# EPICS substitutions: src/main/epics/hnossApp/Db/hnoss.substitutions
#HNOSS

file "DI.template" { pattern

#PSL SUBS?
{SUBS,	DEV,       OFFS,   OFFS2}
{Rhtr,	LS550,      84,	    84}
{PSL,	PSL,        86,     86}
}

file "AI.template" { pattern

#unsure about units..
{SUBS,	DEV,       OFFS,   OFFS2, LOPR, HOPR, EGU}
{LHe,	TT140A,   130,	   130,	  0,	500,   K}
{LHe,	TT140B,   136,	   136,	  0,	500,   K}
{LHe,   TT140C,   142,     142,   0,    500,   K}
{LHe,   TT140D,   148,     148,   0,    500,   K}
{LHe,   TT141,    154,     154,   0,    500,   K}
{LHe,   TT142A,   160,     160,   0,    500,   K}
{LHe,   TT142B,   166,     166,   0,    500,   K}
{LHe,   TT143A,   172,     172,   0,    500,   K}
{LHe,   TT143B,   178,     178,   0,    500,   K}
{LHe,   TT143C,   184,     184,   0,    500,   K}
{LHe,   TT144A,   190,     190,   0,    500,   K}
{LHe,   TT144B,   196,     196,   0,    500,   K}
{LHe,   TT144C,   202,     202,   0,    500,   K}
{LHe,   TT145A,   208,     208,   0,    500,   K}
{LHe,   TT145B,   214,     214,   0,    500,   K}
{LHe,   TT146A,   220,     220,   0,    500,   K}
{LHe,   TT146B,   226,     226,   0,    500,   K}
{LHe,   TT147,    232,     232,   0,    500,   K}
{LHe,   TT148,    238,     238,   0,    500,   K}
{LN2,   TT200,    244,     244,   0,    500,   K}
{LN2,   TT201,    250,     250,   0,    500,   K}
{LN2,   TT202,    256,     256,   0,    500,   K}
{LN2,   TT203,    262,     262,   0,    500,   K}
{LN2,   TT204,    268,     268,   0,    500,   K}
{LN2,   TT205,    274,     274,   0,    500,   K}
{LN2,   TT206,    280,     280,   0,    500,   K}
{LN2,   TT207,    286,     286,   0,    500,   K}
{LN2,   TT208,    292,     292,   0,    500,   K}
{LN2,   TT209,    298,     298,   0,    500,   K}
{LN2,   TT210,    304,     304,   0,    500,   K}
{LN2,   TT211,    310,     310,   0,    500,   K}
{LN2,   TT212,    316,     316,   0,    500,   K}
{LN2,   TT213,    322,     322,   0,    500,   K}
{LN2,   TT214A,   328,     328,   0,    500,   K}
{LN2,   TT214B,   334,     334,   0,    500,   K}
{LN2,   TT214C,   340,     340,   0,    500,   K}
{LN2,   TT215,    346,     346,   0,    500,   K}
{LN2,   TT216A,   352,     352,   0,    500,   K}
{LN2,   TT216B,   358,     358,   0,    500,   K}
{LN2,   TT216C,   364,     364,   0,    500,   K}
{LN2,   TT216D,   370,     370,   0,    500,   K}
{LN2,   TT216E,   376,     376,   0,    500,   K}
{LN2,   TT216F,   382,     382,   0,    500,   K}
{LN2,   TT217,    388,     388,   0,    500,   K}
{SHe,   TT300,    394,     394,   0,    500,   K}
{SHe,   TT307,    400,     400,   0,    500,   K}
{SHe,   TT308,    406,     406,   0,    500,   K}
{SHe,   TT309,    412,     412,   0,    500,   K}
{SHe,   TT310,    418,     418,   0,    500,   K}
{SHe,   TT311,    424,     424,   0,    500,   K}
{SHe,   TT312,    430,     430,   0,    500,   K}
{IBoxN2,TT400,    436,     436,   0,    500,   K}
{IBoxN2,TT401A,   442,     442,   0,    500,   K}
{IBoxN2,TT401B,   448,     448,   0,    500,   K}
{IBoxN2,TT401C,   454,     454,   0,    500,   K}
{IBoxN2,TT402,    460,     460,   0,    500,   K}
{IBoxN2,TT403,    466,     466,   0,    500,   K}
{IBoxN2,TT404,    472,     472,   0,    500,   K}
{IBoxN2,TT405,    478,     478,   0,    500,   K}
{RHtr,  TT550,    484,     484,   0,    500,   K}
{SHe,   PT300,    490,     490,   0,    500,   Pa}
{SHe,   PT301,    496,     496,   0,    500,   Pa}
{SHe,   PT302,    502,     502,   0,    500,   Pa}
{IBoxHe,PT500,    508,     508,   0,    500,   Pa}
{LN2,   PT200,    514,     514,   0,    500,   Pa}
{LHe,   LT100,    520,     520,   0,    500,   m}
{LHe,   LT101,    526,     526,   0,    500,   m}
{LN2,   FT200,    532,     532,   0,    500,   m3/s}
{LN2,   FT201,    538,     538,   0,    500,   m3/s}
{LN2,   FT202,    544,     544,   0,    500,   m3/s}
{SHe,   FT301,    550,     550,   0,    500,   m3/s}
{SHe,   FT302,    556,     556,   0,    500,   m3/s}
{RHtr,  FT550,    562,     562,   0,    500,   m3/s}
{RHtr,  FT551,    568,     568,   0,    500,   m3/s}
{RHtr,  FT552,    574,     574,   0,    500,   m3/s}
{LHe,   TT100,    706,     706,   0,    500,   K}
{LHe,   TT101,    712,     712,   0,    500,   K}
{LHe,   TT102,    718,     718,   0,    500,   K}
{LHe,   TT103,    724,     724,   0,    500,   K}
{LHe,   TT104,    730,     730,   0,    500,   K}
{LHe,   TT105,    736,     736,   0,    500,   K}
{LHe,   TT106,    742,     742,   0,    500,   K}
{LHe,   TT107,    748,     748,   0,    500,   K}
{LHe,   TT108,    754,     754,   0,    500,   K}
{LHe,   TT109,    760,     760,   0,    500,   K}
{LHe,   TT110,    766,     766,   0,    500,   K}
{LHe,   TT111,    772,     772,   0,    500,   K}
{LHe,   TT112,    778,     778,   0,    500,   K}
{LHe,   TT113,    784,     784,   0,    500,   K}
{LHe,   TT114,    790,     790,   0,    500,   K}
{LHe,   TT115,    796,     796,   0,    500,   K}
{LHe,   TT116,    802,     802,   0,    500,   K}
{LHe,   TT117,    808,     808,   0,    500,   K}
{LHe,   TT118,    814,     814,   0,    500,   K}
{LHe,   TT119,    820,     820,   0,    500,   K}
{LHe,   TT120,    826,     826,   0,    500,   K}
{LHe,   TT121,    832,     832,   0,    500,   K}
{LHe,   TT122,    838,     838,   0,    500,   K}
{LHe,   TT123,    844,     844,   0,    500,   K}
{LHe,   TT124,    850,     850,   0,    500,   K}
{LHe,   TT125,    856,     856,   0,    500,   K}
{LHe,   TT126,    862,     862,   0,    500,   K}
{LHe,   TT127,    868,     868,   0,    500,   K}
{LHe,   TT128,    874,     874,   0,    500,   K}
{LHe,   TT129,    880,     880,   0,    500,   K}
{LHe,   TT130,    886,     886,   0,    500,   K}
{SHe,   TT301,    892,     892,   0,    500,   K}
{SHe,   TT302,    898,     898,   0,    500,   K}
{SHe,   TT303,    904,     904,   0,    500,   K}
{SHe,   TT304,    910,     910,   0,    500,   K}
{SHe,   TT305,    916,     916,   0,    500,   K}
{SHe,   TT306,    922,     922,   0,    500,   K}
{IBoxHe,TT500,    928,     928,   0,    500,   K}
{IBoxHe,TT501,    934,     934,   0,    500,   K}
{IBoxHe,TT502,    940,     940,   0,    500,   K}
{RHtr,  PT551,   1072,    1072,   0,    500,   Pa}
{RHtr,  PT552,   1078,    1078,   0,    500,   Pa}
{LHe,   PT100,   1084,    1084,   0,    500,   Pa}
{RHtr,  PT550,   1090,    1090,   0,    500,   Pa}
{LHe,   PT101,   1096,    1096,   0,    500,   Pa}
{LHe,   PT102,   1102,    1102,   0,    500,   Pa}
{Vac,   PT000,   1234,    1234,   0,    500,   Pa}
{Vac,   PT001,   1240,    1240,   0,    500,   Pa}
{Vac,   PT002,   1246,    1246,   0,    500,   Pa}
{Vac,   PT003,   1252,    1252,   0,    500,   Pa}
{Vac,   PT004,   1258,    1258,   0,    500,   Pa}
}

file "Valves.template" { pattern
{SUBS,	DEV,       OFFS,   OFFS2}
{Vac,	FV000,     1438,    1438}
{Vac,	FV001,     1440,    1440}
{Vac,	FV010,     1442,    1442}
{Vac,	FV011,     1444,    1444}
{Vac,	FV012,     1446,    1446}
{LHe,	FV100,     1448,    1448}
{LHe,	FV101,     1450,    1450}
{LN2,	FV200,     1452,    1452}
{SHe,	FV300,     1454,    1454}
{SHe,	FV301,     1456,    1456}
{SHe,	FV302,     1458,    1458}
{IBoxN2,FV400,     1460,    1460}
{IBoxN2,FV401,     1462,    1462}
{IBoxHe,FV500,     1464,    1464}
{IBoxHe,FV501,     1466,    1466}
{IBoxHe,FV502,     1468,    1468}
{RHtr,  FV550,     1470,    1470}
{RHtr,  FV551,     1472,    1472}
}

file "Evalves.template" { pattern
{SUBS,	DEV,       OFFS,   OFFS2}
{LN2,	EV200,     1390,    1390}
{LN2,	EV201,     1392,    1392}
{IBoxN2,EV400,     1394,    1394}
}

file "AValves.template" { pattern
{SUBS,	DEV,       OFFS,   OFFS2, LOPR, HOPR, EGU}
{LHe,	CV100,   1516,	   1516,   0,	100,  percent}
{LHe,	CV101,   1522,	   1522,   0,	100,  percent}
{LHe,	CV102,   1528,	   1528,   0,	100,  percent}
{LHe,	CV103,   1534,	   1534,   0,	100,  percent}
{LHe,	CV104,   1540,	   1540,   0,	100,  percent}
{LHe,	CV105,   1546,	   1546,   0,	100,  percent}
{LN2,	CV200,   1552,	   1552,   0,	100,  percent}
{LN2,	CV201,   1558,	   1558,   0,	100,  percent}
{SHe,	CV301,   1564,	   1564,   0,	100,  percent}
{SHe,	CV302,   1570,	   1570,   0,	100,  percent}
{RHtr,	CV550,   1576,	   1576,   0,	100,  percent}
{RHtr,	CV551,   1582,	   1582,   0,	100,  percent}
{RHtr,	CV552,   1588,	   1588,   0,	100,  percent}
}

file "PID.template" { pattern
{SUBS,   DEV,     OFFS,   OFFS2,    EGU}
{LN2,    TIC200,  1720,   1720,    unknown}
{LN2,    FIC200,  1742,   1730,    unknown}
{LN2,    TIC201,  1764,   1740,    unknown}
{LN2,    FIC201,  1786,   1750,    unknown}
{SHe,    TIC301,  1808,   1760,    unknown}
{SHe,    FIC301,  1830,   1770,    unknown}
{SHe,    TIC302,  1852,   1780,    unknown}
{SHe,    FIC302,  1874,   1790,    unknown}
{LHe,    TIC101,  1896,   1800,    unknown}
{MKS,    MKS1,    1918,   1810,    unknown}
{MKS,    MKS2,    1940,   1820,    unknown}
{MKS,    MKS3,    1962,   1830,    unknown}
}

file "Heater1.template" { pattern
{SUBS,	DEV,       OFFS,   OFFS2}
{LHe,	EH100,     2446,    2050}
{LHe,	EH101,     2456,    2060}
{LHe,	EH102,     2466,    2070}
{LHe,	EH103,     2476,    2080}
{LHe,	EH104,     2486,    2090}
{LHe,	EH105,     2496,    2100}
{LHe,	EH106,     2506,    2110}
{LHe,	EH107,     2516,    2120}
{LHe,	EH108,     2526,    2130}
{LN2,	EH200,     2536,    2140}
{LN2,	EH201,     2546,    2150}
{LN2,	EH202,     2556,    2160}
{LN2,	EH203,     2566,    2170}
{LN2,	EH204,     2576,    2180}
{LN2,	EH205,     2586,    2190}
{LN2,	EH206,     2596,    2200}
{LN2,	EH207,     2606,    2210}
{LN2,	EH208,     2616,    2220}
{SHe,	EH300,     2626,    2230}
{SHe,	EH301,     2636,    2240}
{SHe,	EH302,     2646,    2250}
{SHe,	EH303,     2656,    2260}
{IBoxN2,EH400,     2666,    2270}
{IBoxN2,EH401,     2676,    2280}
}

file "Heater2.template" { pattern
{SUBS,	DEV,       OFFS,   OFFS2}
{Rhtr,	EH550,     2896,    2500}
}

file "SQbinary.template" { pattern
{SUBS, OFFS2, OFFS}
{SQ0,   2808, 3204}
{SQ1,   2892, 3306}
{SQ2,   2976, 3408}
{SQ3A,  3060, 3510}
{SQ3B,  3144, 3612}
{SQ4,   3228, 3714}
{SQ5,   3312, 3816}
{SQ6,   3396, 3918}
{SQ7,   3480, 4020}
{SQ8,   3564, 4122}
{SQ9,   3648, 4224}
{SQ10,  3732, 4326}
{SQ11,  3816, 4428}
{SQ12A, 3900, 4530}
{SQ12B, 3984, 4632}
{SQ13,  4068, 4734}
{SQ20,  4152, 4836}
}

file "SQanalog.template" { pattern
{SUBS,	 SIG,          OFFS2, TYPE, SIG2,	OFFS, EGU}
{SQ0,	cNcycle,       2810, INT16, sNcycle, 3224, ""}
{SQ0,	cVacRate,      2812, INT16, sVacRate, 3226,	"s"}
{SQ0,	cPressRate,    2814, INT16, sPressRate, 3228,	"s"}
{SQ0,	cVacRateAlrm,  2816, INT16, sVacRateAlrm, 3230,	"s"}
{SQ0,	cPresRateAlrm, 2818, INT16, sPresRateAlrm, 3232,"s"}
{SQ0,	cVac,          2828, FLOAT, sVac, 3242,	   "mbar"}
{SQ0,	cVacFlt,       2832, FLOAT, sVacFlt, 3246, "mbar"}
{SQ0,	cPressEOF,     2836, FLOAT, sPressEOF, 3250, "mbar"}
{SQ0,	cPressFlt,     2840, FLOAT, sPressFlt, 3254, "mbar"}
{SQ1,	cNcycle,       2894, INT16, sNcycle, 3326,   ""}
{SQ1,	cVacRate,      2896, INT16, sVacRate, 3328,  "s"}
{SQ1,	cPressRate,    2898, INT16, sPressRate, 3330,	"s"}
{SQ1,	cVacRateAlrm,  2900, INT16, sVacRateAlrm, 3332,	"s"}
{SQ1,	cPresRateAlrm, 2902, INT16, sPresRateAlrm, 3334,	"s"}
{SQ1,	cVac,          2912, FLOAT, sVac, 3344,	   "mbar"}
{SQ1,	cVacFlt,       2916, FLOAT, sVacFlt, 3348,	   "mbar"}
{SQ1,	cPressEOF,     2920, FLOAT, sPressEOF, 3352,	   "mbar"}
{SQ1,	cPressFlt,     2924, FLOAT, sPressFlt, 3356,	   "mbar"}
{SQ1,	cP_CV100,      2928, FLOAT, sP_CV100, 3360,   ""}
{SQ1,	cP_CV101,      2932, FLOAT, sP_CV101, 3364,   ""}
{SQ1,	cP_CV102,      2936, FLOAT, sP_CV102, 3368,   ""}
{SQ1,	cP_CV103,      2940, FLOAT, sP_CV103, 3372,   ""}
{SQ1,	cP_CV104,      2944, FLOAT, sP_CV104, 3376,   ""}
{SQ1,	cP_CV105,      2948, FLOAT, sP_CV105, 3380,   ""}
{SQ1,	cP_CV550,      2952, FLOAT, sP_CV550, 3384,   ""}
{SQ1,	cP_CV551,      2956, FLOAT, sP_CV551, 3388,   ""}
{SQ2,	cNcycle,       2978, INT16, sNcycle, 3428,   ""}
{SQ2,	cVacRate,      2980, INT16, sVacRate, 3430	"s"}
{SQ2,	cPressRate,    2982, INT16, sPressRate, 3432	"s"}
{SQ2,	cVacRateAlrm,  2984, INT16, sVacRateAlrm, 3434	"s"}
{SQ2,	cPresRateAlrm, 2986, INT16, sPresRateAlrm, 3436	"s"}
{SQ2,	cVac,          2996, FLOAT, sVac, 3446	"mbar"}
{SQ2,	cVacFlt,       3000, FLOAT, sVacFlt, 3450	"mbar"}
{SQ2,	cPressEOF,     3004, FLOAT, sPressEOF, 3454	"mbar"}
{SQ2,	cPressFlt,     3008, FLOAT, sPressFlt, 3458	"mbar"}
{SQ2,	cP_CV301,      3012, FLOAT, sP_CV301, 3462	""}
{SQ2,	cP_CV302,      3016, FLOAT, sP_CV302, 3466	""}
{SQ3A,	cP_Tt,         3080, FLOAT, sP_Tt, 3548	""}
{SQ3A,	cP_Low_Tt,     3084, FLOAT, sP_Low_Tt, 3552	""}
{SQ3A,	cP_High_Tt,    3088, FLOAT, sP_High_Tt, 3556	""}
{SQ3B,	cP_Tt,         3164, FLOAT, sP_Tt, 3650	""}
{SQ3B,	cP_Low_Tt,     3168, FLOAT, sP_Low_Tt, 3654	""}
{SQ3B,	cP_High_Tt,    3172, FLOAT, sP_High_Tt, 3658	""}
{SQ4,	cP_CV200_Tt,   3248, FLOAT, sP_CV200_Tt, 3752	""}
{SQ4,	cP_CV200_Ft,   3252, FLOAT, sP_CV200_Ft, 3756	""}
{SQ4,	cP_CV201_Tt,   3256, FLOAT, sP_CV201_Tt, 3760	""}
{SQ4,	cP_CV201_Ft,   3260, FLOAT, sP_CV201_Ft, 3764	""}
{SQ5,	cP_PT,         3332,  FLOAT, sP_PT,      3854	""}
{SQ5,	cP_FT,         3336,  FLOAT, sP_FT,      3858	""}
{SQ5,	cP_CV550,      3340,  FLOAT, sP_CV550,   3862	""}
{SQ5,	cP_LowLt,      3344,  FLOAT, sP_LowLt,   3866	""}
{SQ5,	cP_CoolD_Tt,   3348,  FLOAT, sP_CoolD_Tt,3870	""}
{SQ5,	cP_HighLt,     3352,  FLOAT, sP_HighLt,  3874	""}
{SQ5,	cP_CV100,      3356,  FLOAT, sP_CV100,   3878	""}
{SQ6,	cP_Tt,         3416,  FLOAT, sP_Tt,      3956	""}
{SQ6,	cP_Lt,         3420,  FLOAT, sP_Lt,      3960	""}
{SQ7,	cP_PT,         3500,  FLOAT, sP_PT,      4058	""}
{SQ7,	cP_FT550,      3504,  FLOAT, sP_FT550,   4062	""}
{SQ7,	cP_Tt_Cold,    3508,  FLOAT, sP_Tt_Cold, 4066	""}
{SQ7,	cP_SP_Tt,      3512,  FLOAT, sP_SP_Tt,   4070	""}
{SQ7,	cP_CV550,      3516,  FLOAT, sP_CV550,   4074	""}
{SQ7,	cP_CV551,      3520,  FLOAT, sP_CV551,   4078	""}
{SQ7,	cP_FT552,      3524,  FLOAT, sP_FT552,   4082	""}
{SQ7,	cP_HighLt,     3528,  FLOAT, sP_HighLt,  4086	""}
{SQ7,	cP_LowLt,      3532,  FLOAT, sP_LowLt,   4090	""}
{SQ7,	cP_CV552,      3536,  FLOAT, sP_CV552,   4094	""}
{SQ7,	cP_CV101,      3540,  FLOAT, sP_CV101,   4098	""}
{SQ7,	cP_CV102,      3544,  FLOAT, sP_CV102,   4102	""}
{SQ7,	cP_CV103,      3548,  FLOAT, sP_CV103,   4106	""}
{SQ7,	cP_CV104,      3552,  FLOAT, sP_CV104,   4110	""}
{SQ8,	cP_CV550,      3584,  FLOAT, sP_CV550,   4160	""}
{SQ8,	cP_LowLt,      3588,  FLOAT, sP_LowLt,   4164	""}
{SQ8,	cP_HighLt,     3592,  FLOAT, sP_HighLt,  4168	""}
{SQ8,	cP_Pt,         3596,  FLOAT, sP_Pt,      4172	""}
{SQ8,	cP_SP_Tt,      3600,  FLOAT, sP_SP_Tt,   4176	""}
{SQ8,	cP_CV551,      3604,  FLOAT, sP_CV551,   4180	""}
{SQ8,	cP_CV552,      3608,  FLOAT, sP_CV552,   4184	""}
{SQ8,	cP_CV104,      3612,  FLOAT, sP_CV104,   4188	""}
{SQ9,	cP_CV550,      3668,  FLOAT, sP_CV550,   4262	""}
{SQ9,	cP_LowLt,      3672,  FLOAT, sP_LowLt,   4266	""}
{SQ9,	cP_HighLt,     3676,  FLOAT, sP_HighLt,  4270	""}
{SQ9,	cP_Pt,         3680,  FLOAT, sP_Pt,      4274	""}
{SQ9,	cP_SP_Tt,      3684,  FLOAT, sP_SP_Tt,   4278	""}
{SQ9,	cP_CV105,      3688,  FLOAT, sP_CV105,   4282	""}
{SQ9,	cP_CV551_Reg,  3692,  FLOAT, sP_CV551_Reg,4286	""}
{SQ9,	cP_Final_Pt,   3696,  FLOAT, sP_Final_Pt,4290	""}
{SQ9,	cP_CV551_Pt00, 4740,  FLOAT, sP_CV551_Pt00,5550	""}
{SQ9,	cP_CV551_Pt01, 4744,  FLOAT, sP_CV551_Pt01,5554	""}
{SQ9,	cP_CV551_Pt02, 4748,  FLOAT, sP_CV551_Pt02,5558	""}
{SQ9,	cP_CV551_Pt03, 4752,  FLOAT, sP_CV551_Pt03,5562	""}
{SQ9,	cP_CV551_Pt04, 4756,  FLOAT, sP_CV551_Pt04,5566	""}
{SQ9,	cP_CV551_Pt05, 4760,  FLOAT, sP_CV551_Pt05,5570	""}
{SQ9,	cP_CV551_Pt06, 4764,  FLOAT, sP_CV551_Pt06,5574	""}
{SQ9,	cP_CV551_Pt07, 4768,  FLOAT, sP_CV551_Pt07,5578	""}
{SQ9,	cP_CV551_Pt08, 4772,  FLOAT, sP_CV551_Pt08,5582	""}
{SQ9,	cP_CV551_Pt09, 4776,  FLOAT, sP_CV551_Pt09,5586	""}
{SQ9,	cP_CV551_Pt10, 4780,  FLOAT, sP_CV551_Pt10,5590	""}
{SQ9,	cP_CV551_Pt11, 4784,  FLOAT, sP_CV551_Pt11,5594	""}
{SQ9,	cP_CV551_Pt12, 4788,  FLOAT, sP_CV551_Pt12,5598	""}
{SQ9,	cP_CV551_Csg00, 4804,  FLOAT, sP_CV551_Csg00,5614	""}
{SQ9,	cP_CV551_Csg01, 4808,  FLOAT, sP_CV551_Csg01,5618	""}
{SQ9,	cP_CV551_Csg02, 4812,  FLOAT, sP_CV551_Csg02,5622	""}
{SQ9,	cP_CV551_Csg03, 4816,  FLOAT, sP_CV551_Csg03,5626	""}
{SQ9,	cP_CV551_Csg04, 4820,  FLOAT, sP_CV551_Csg04,5630	""}
{SQ9,	cP_CV551_Csg05, 4824,  FLOAT, sP_CV551_Csg05,5634	""}
{SQ9,	cP_CV551_Csg06, 4828,  FLOAT, sP_CV551_Csg06,5638	""}
{SQ9,	cP_CV551_Csg07, 4832,  FLOAT, sP_CV551_Csg07,5642	""}
{SQ9,	cP_CV551_Csg08, 4836,  FLOAT, sP_CV551_Csg08,5646	""}
{SQ9,	cP_CV551_Csg09, 4840,  FLOAT, sP_CV551_Csg09,5650	""}
{SQ9,	cP_CV551_Csg10, 4844,  FLOAT, sP_CV551_Csg10,5654	""}
{SQ9,	cP_CV551_Csg11, 4848,  FLOAT, sP_CV551_Csg11,5658	""}
{SQ9,	cP_CV551_Csg12, 4852,  FLOAT, sP_CV551_Csg12,5662	""}
{SQ10,	cP_CV301_Tt,   3752,  FLOAT, sP_CV301_Tt,4364	""}
{SQ10,	cP_CV301_Ft,   3756,  FLOAT, sP_CV301_Ft,4368	""}
{SQ10,	cP_CV302_Tt,   3760,  FLOAT, sP_CV302_Tt,4372	""}
{SQ10,	cP_CV302_Ft,   3764,  FLOAT, sP_CV302_Ft,4376	""}
{SQ11,	cP_CV550,      3836,  FLOAT, sP_CV550,   4466	""}
{SQ11,	cP_Tt,         3840,  FLOAT, sP_Tt,      4470	""}
{SQ11,	cP_Pt,         3844,  FLOAT, sP_Pt, 	 4474	""}
{SQ11,	cP_SP_Tt,      3848,  FLOAT, sP_SP_Tt,   4478	""}
{SQ11,	cP_CV551,      3852,  FLOAT, sP_CV551,   4482	""}
{SQ11,	cP_CV552,      3856,  FLOAT, sP_CV552,   4486	""}
{SQ11,	cP_CV104,      3860,  FLOAT, sP_CV104,   4490	""}
{SQ12A,	cP_WarmUp,     3920,  FLOAT, sP_WarmUp,  4568	""}
{SQ12B,	cP_WarmUp,     4004,  FLOAT, sP_WarmUp,  4670	""}
{SQ12B,	cP_CV550,      4008,  FLOAT, sP_CV550,   4674	""}
{SQ12B,	cP_CV551,      4012,  FLOAT, sP_CV551,   4678	""}
{SQ12B,	cP_CV552,      4016,  FLOAT, sP_CV552,   4682	""}
{SQ12B,	cP_CV100,      4020,  FLOAT, sP_CV100,   4686	""}
{SQ12B,	cP_CV101,      4024,  FLOAT, sP_CV101,   4690	""}
{SQ12B,	cP_CV102,      4028,  FLOAT, sP_CV102,   4694	""}
{SQ12B,	cP_CV103,      4032,  FLOAT, sP_CV103,   4698	""}
{SQ12B,	cP_CV104,      4036,  FLOAT, sP_CV104,   4702	""}
{SQ12B,	cP_CV105,      4040,  FLOAT, sP_CV105,   4706	""}
{SQ12B,	cP_CV200,      4044,  FLOAT, sP_CV200,   4710	""}
{SQ12B,	cP_CV201,      4048,  FLOAT, sP_CV201,   4714	""}
{SQ12B,	cP_CV302,      4052,  FLOAT, sP_CV302,   4718	""}
{SQ12B,	cP_CV301,      4056,  FLOAT, sP_CV301,   4722	""}
{SQ13,	cP_Al_SHe,     4088,  FLOAT, sP_Al_SHe,  4772	""}
{SQ13,	cP_Al_He,      4092,  FLOAT, sP_Al_He,   4776	""}
{SQ13,	cP_SHe,        4096,  FLOAT, sP_SHe,   	 4780	""}
{SQ13,	cP_He,         4100,  FLOAT, sP_He,   	 4784	""}
{SQ20,	cP_Op,         4154,  INT16, sP_Op,   	 4856	""}
}

file "SQbinPar.template" { pattern
{SUBS,	 SIG,          OFFS2, BIT2, OFFS, BIT}
{SQ4,	 P_C1,          3229, 0,    3732, 0}
{SQ4,	 P_C2,          3229, 1,    3732, 1}
{SQ4,	 P_Tt,          3229, 2,    3732, 2}
{SQ4,	 P_Ft,          3229, 3,    3732, 3}
{SQ7,	 P_C1,          3481, 0,    4038, 0}
{SQ7,	 P_C2,          3481, 1,    4038, 1}
{SQ7,	 P_Tbl,         3481, 2,    4038, 2}
{SQ7,	 P_MS,          3481, 3,    4038, 3}
{SQ8,	 P_MS,          3565, 0,    4140, 0}
{SQ8,	 P_Tbl,         3565, 1,    4140, 1}
{SQ9,	 P_MS,          3649, 0,    4242, 0}
{SQ9,	 P_Tbl,         3649, 1,    4242, 1}
{SQ10,	 P_C1,          3733, 0,    4344, 0}
{SQ10,	 P_C2,          3733, 1,    4344, 1}
{SQ10,	 P_Tt,          3733, 2,    4344, 2}
{SQ10,	 P_Ft,          3733, 3,    4344, 3}
{SQ11,	 P_MS,          3817, 0,    4446, 0}
{SQ11,	 P_Tbl,         3817, 1,    4446, 1}
{SQ13,	 P_Isolated,    4069, 0,    4752, 0}
{SQ20,	 P_CondCryo,    4153, 0,    4854, 0}
{SQ20,	 P_CondCoupl,   4153, 1,    4854, 1}
{SQ20,	 P_CDCryo,      4153, 2,    4854, 2}
{SQ20,	 P_SHe,         4153, 3,    4854, 3}
{SQ20,	 P_WarmUp,      4153, 4,    4854, 4}
{SQ20,	 P_Isolated,    4153, 5,    4854, 5}
{SQ20,	 P_StopSeq,     4153, 6,    4854, 6}
}

file "SQ0_1_2.template" { pattern
{SUBS, OFFS}
{SQ0, 3205}
{SQ1, 3307}
{SQ2, 3409}
}
